ABB RobotStudio station: simulation.rsstn

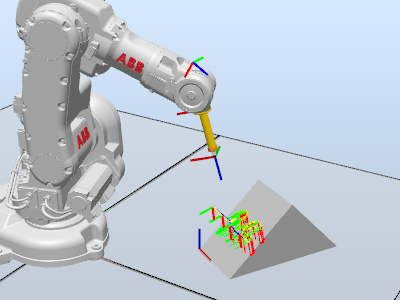
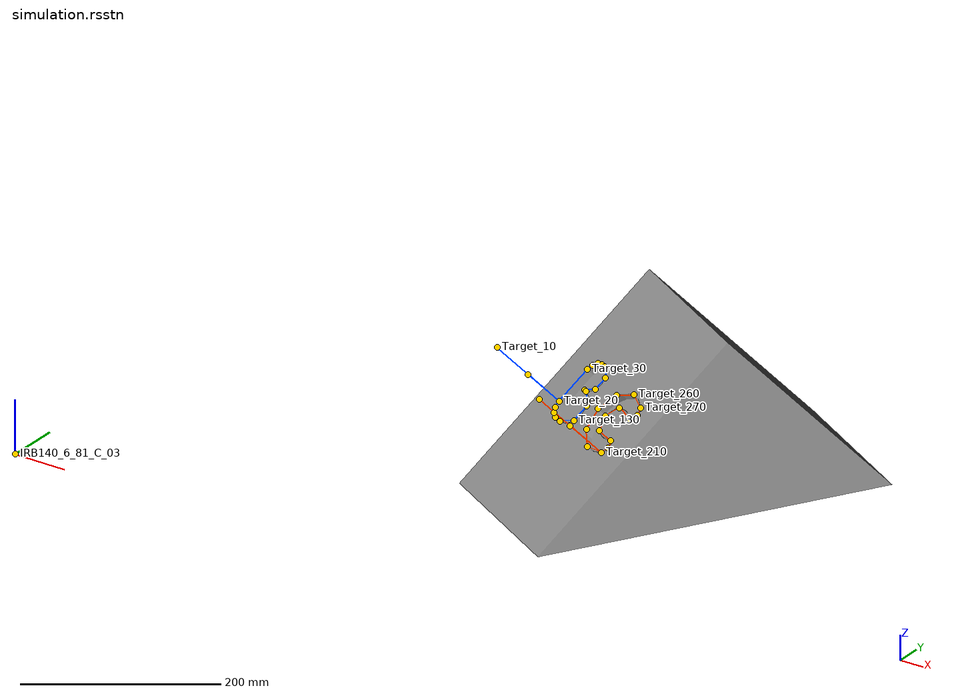
[picture v1: parts stored in the station drawn from their meshes, with robot base, taught points and paths (robot models come from the ABB library and are not in the file)]
Station simulation (saved by RobotStudio 22.2.9947.0)
Controller Controller7
  mechanical unit ROB_1: IRB140_6_81_C_03, 6 joints, base frame (0, 0, 0) mm
Layout (positions relative to the parent item):
  - IRB140_6_81_C_03 [mechanism, from Robots\IRB140_6_81_C_G_03.rslib] at (0, 0, 0) mm; joint values [0.3491, 0.0873, 0.3491, 0, 0.8727, 0] (rad or m)
  - MarkerTool [mechanism] at (434.7, 158.22, 487.25) mm, rotated rx 180 ry 15 rz -160 deg
      TCP MarkerTool at (0, 0, 145) mm
      links: ToolAssambly
  - Triangle [part] at (400, 200, 0) mm, rotated rx 0 ry 0 rz -30 deg, size 185 x 389.2 x 194.1 mm
Attachment: MarkerTool is attached to IRB140_6_81_C_03 / Link6
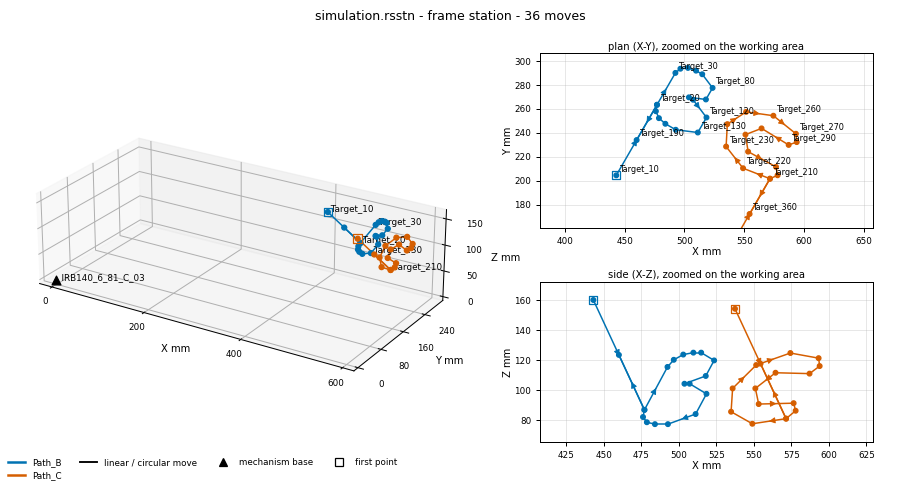
[picture p0: tool path of simulation.rsstn in frame station, 36 of 38 moves have a stored position in this frame; points joined in program order, loops and branches not executed]
Targets, tools, work objects and paths stored in the station, written as RAPID:
! task T_ROB1
MODULE CalibData
  PERS tooldata MarkerTool:=[TRUE,[[0,0,145],[1,0,0,0]],[0.1,[0,0,61],[1,0,0,0],0,0,0]];
  TASK PERS wobjdata Canvas:=[FALSE,TRUE,"",[[400.001,200,0],[0.9659258,0,0,-0.258819143]],[[0,0,0],[1,0,0,0]]];
ENDMODULE

! task T_ROB1
MODULE Module1
  CONST robtarget Target_10:=[[34.950823156,25.414242905,160.180640129],[0.35336537,-0.898969249,0.240877877,0.094683961],[0,0,0,0],[9E+09,9E+09,9E+09,9E+09,9E+09,9E+09]];
  CONST robtarget Target_20:=[[34.950809352,93.508617436,86.947067519],[0.35336537,-0.898969249,0.240877877,0.094683961],[0,0,0,0],[9E+09,9E+09,9E+09,9E+09,9E+09,9E+09]];
  CONST robtarget Target_30:=[[34.950803116,124.266717933,115.546704822],[0.35336537,-0.898969249,0.240877877,0.094683961],[0,0,0,0],[9E+09,9E+09,9E+09,9E+09,9E+09,9E+09]];
  CONST robtarget Target_40:=[[36.826446423,129.393068396,120.31331104],[0.353365369,-0.89896925,0.240877877,0.094683961],[0,0,0,0],[9E+09,9E+09,9E+09,9E+09,9E+09,9E+09]];
  CONST robtarget Target_50:=[[41.950801316,133.145818152,123.80270897],[0.35336537,-0.898969249,0.240877877,0.09468396],[0,0,0,0],[9E+09,9E+09,9E+09,9E+09,9E+09,9E+09]];
  CONST robtarget Target_60:=[[48.950801037,134.519420935,125.079917257],[0.35336537,-0.898969249,0.240877877,0.094683961],[0,0,0,0],[9E+09,9E+09,9E+09,9E+09,9E+09,9E+09]];
  CONST robtarget Target_70:=[[54.950801037,134.519422152,125.079917257],[0.35336537,-0.898969249,0.240877877,0.094683961],[0,0,0,0],[9E+09,9E+09,9E+09,9E+09,9E+09,9E+09]];
  CONST robtarget Target_80:=[[68.129449616,128.947305169,119.898823543],[0.35336537,-0.898969249,0.240877877,0.094683961],[0,0,0,0],[9E+09,9E+09,9E+09,9E+09,9E+09,9E+09]];
  CONST robtarget Target_90:=[[68.129451875,117.803065859,109.536636114],[0.353365369,-0.89896925,0.240877877,0.094683961],[0,0,0,0],[9E+09,9E+09,9E+09,9E+09,9E+09,9E+09]];
  CONST robtarget Target_100:=[[54.950805555,112.230943533,104.355542399],[0.35336537,-0.898969249,0.240877877,0.094683961],[0,0,0,0],[9E+09,9E+09,9E+09,9E+09,9E+09,9E+09]];
  CONST robtarget Target_110:=[[58.950805555,112.230944343,104.355542399],[0.35336537,-0.898969249,0.240877877,0.094683961],[0,0,0,0],[9E+09,9E+09,9E+09,9E+09,9E+09,9E+09]];
  CONST robtarget Target_120:=[[76.083048708,104.987192264,97.620120571],[0.35336537,-0.898969249,0.240877877,0.094683961],[0,0,0,0],[9E+09,9E+09,9E+09,9E+09,9E+09,9E+09]];
  CONST robtarget Target_130:=[[76.083051645,90.499681161,84.149276913],[0.353365369,-0.89896925,0.240877877,0.094683961],[0,0,0,0],[9E+09,9E+09,9E+09,9E+09,9E+09,9E+09]];
  CONST robtarget Target_140:=[[58.95081143,83.255922137,77.413855085],[0.35336537,-0.898969249,0.240877877,0.094683961],[0,0,0,0],[9E+09,9E+09,9E+09,9E+09,9E+09,9E+09]];
  CONST robtarget Target_150:=[[48.95081143,83.25592011,77.413855085],[0.35336537,-0.898969249,0.240877877,0.094683961],[0,0,0,0],[9E+09,9E+09,9E+09,9E+09,9E+09,9E+09]];
  CONST robtarget Target_160:=[[41.950811151,84.629520055,78.691063371],[0.35336537,-0.898969249,0.240877877,0.094683961],[0,0,0,0],[9E+09,9E+09,9E+09,9E+09,9E+09,9E+09]];
  CONST robtarget Target_170:=[[36.826454737,88.382267733,82.180461302],[0.35336537,-0.898969249,0.240877877,0.094683961],[0,0,0,0],[9E+09,9E+09,9E+09,9E+09,9E+09,9E+09]];
  CONST robtarget Target_180:=[[34.950809352,93.508617436,86.947067519],[0.35336537,-0.898969249,0.240877877,0.094683961],[0,0,0,0],[9E+09,9E+09,9E+09,9E+09,9E+09,9E+09]];
  CONST robtarget Target_190:=[[34.950816254,59.461430171,123.563853824],[0.35336537,-0.898969249,0.240877877,0.094683961],[0,0,0,0],[9E+09,9E+09,9E+09,9E+09,9E+09,9E+09]];
  CONST robtarget Target_200:=[[147.617491101,19.11128582,154.319974583],[0.35336537,-0.898969249,0.240877877,0.094683961],[0,0,0,0],[9E+09,9E+09,9E+09,9E+09,9E+09,9E+09]];
  CONST robtarget Target_210:=[[147.617477296,87.205660351,81.086401974],[0.35336537,-0.898969249,0.240877877,0.094683961],[0,0,0,0],[9E+09,9E+09,9E+09,9E+09,9E+09,9E+09]];
  CONST robtarget Target_220:=[[123.769810397,83.538318205,77.676421666],[0.35336537,-0.898969249,0.240877877,0.094683961],[0,0,0,0],[9E+09,9E+09,9E+09,9E+09,9E+09,9E+09]];
  CONST robtarget Target_230:=[[102.433503633,92.15845815,85.691643532],[0.35336537,-0.898969249,0.240877877,0.094683961],[0,0,0,0],[9E+09,9E+09,9E+09,9E+09,9E+09,9E+09]];
  CONST robtarget Target_240:=[[93.950806233,108.887679646,101.246886171],[0.35336537,-0.898969249,0.240877877,0.094683961],[0,0,0,0],[9E+09,9E+09,9E+09,9E+09,9E+09,9E+09]];
  CONST robtarget Target_250:=[[102.433496851,125.616904581,116.80212881],[0.35336537,-0.898969249,0.240877877,0.094683961],[0,0,0,0],[9E+09,9E+09,9E+09,9E+09,9E+09,9E+09]];
  CONST robtarget Target_260:=[[123.769800119,134.237053177,124.817350675],[0.353365369,-0.89896925,0.240877877,0.094683961],[0,0,0,0],[9E+09,9E+09,9E+09,9E+09,9E+09,9E+09]];
  CONST robtarget Target_270:=[[147.617468505,130.5697207,121.407370368],[0.35336537,-0.898969249,0.240877877,0.094683961],[0,0,0,0],[9E+09,9E+09,9E+09,9E+09,9E+09,9E+09]];
  CONST robtarget Target_280:=[[151.694170772,124.899768155,116.135308461],[0.35336537,-0.898969249,0.240877877,0.094683961],[0,0,0,0],[9E+09,9E+09,9E+09,9E+09,9E+09,9E+09]];
  CONST robtarget Target_290:=[[147.027505204,119.479259665,111.095187412],[0.35336537,-0.898969249,0.240877877,0.094683962],[0,0,0,0],[9E+09,9E+09,9E+09,9E+09,9E+09,9E+09]];
  CONST robtarget Target_300:=[[120.497500856,120.109201737,111.680928024],[0.35336537,-0.898969249,0.240877877,0.094683961],[0,0,0,0],[9E+09,9E+09,9E+09,9E+09,9E+09,9E+09]];
  CONST robtarget Target_310:=[[111.450806233,108.887683193,101.246886171],[0.35336537,-0.898969249,0.240877877,0.094683961],[0,0,0,0],[9E+09,9E+09,9E+09,9E+09,9E+09,9E+09]];
  CONST robtarget Target_320:=[[120.497505406,97.666168317,90.812844318],[0.35336537,-0.898969249,0.240877877,0.094683961],[0,0,0,0],[9E+09,9E+09,9E+09,9E+09,9E+09,9E+09]];
  CONST robtarget Target_330:=[[147.027509499,98.296121147,91.39858493],[0.353365371,-0.898969249,0.240877877,0.094683961],[0,0,0,0],[9E+09,9E+09,9E+09,9E+09,9E+09,9E+09]];
  CONST robtarget Target_340:=[[151.694177264,92.875614549,86.358463881],[0.35336537,-0.898969249,0.240877877,0.094683961],[0,0,0,0],[9E+09,9E+09,9E+09,9E+09,9E+09,9E+09]];
  CONST robtarget Target_350:=[[147.617477296,87.205660351,81.086401974],[0.35336537,-0.898969249,0.240877877,0.094683961],[0,0,0,0],[9E+09,9E+09,9E+09,9E+09,9E+09,9E+09]];
  CONST robtarget Target_360:=[[147.617484199,53.158473085,117.703188278],[0.35336537,-0.898969249,0.240877877,0.094683961],[0,0,0,0],[9E+09,9E+09,9E+09,9E+09,9E+09,9E+09]];
  CONST jointtarget Home:=[[0,0,0,0,30,0],[9E+09,9E+09,9E+09,9E+09,9E+09,9E+09]];
  CONST jointtarget Middle:=[[20,5,20,0,50,0],[9E+09,9E+09,9E+09,9E+09,9E+09,9E+09]];
  PROC Path_B()
    MoveL Target_10,v200,z50,MarkerTool\WObj:=Canvas;
    MoveL Target_20,v200,z50,MarkerTool\WObj:=Canvas;
    MoveL Target_30,v200,z50,MarkerTool\WObj:=Canvas;
    MoveL Target_40,v200,z50,MarkerTool\WObj:=Canvas;
    MoveL Target_50,v200,z50,MarkerTool\WObj:=Canvas;
    MoveL Target_60,v200,z50,MarkerTool\WObj:=Canvas;
    MoveL Target_70,v200,z50,MarkerTool\WObj:=Canvas;
    MoveL Target_80,v200,z50,MarkerTool\WObj:=Canvas;
    MoveL Target_90,v200,z50,MarkerTool\WObj:=Canvas;
    MoveL Target_100,v200,z50,MarkerTool\WObj:=Canvas;
    MoveL Target_110,v200,z50,MarkerTool\WObj:=Canvas;
    MoveL Target_120,v200,z50,MarkerTool\WObj:=Canvas;
    MoveL Target_130,v200,z50,MarkerTool\WObj:=Canvas;
    MoveL Target_140,v200,z50,MarkerTool\WObj:=Canvas;
    MoveL Target_150,v200,z50,MarkerTool\WObj:=Canvas;
    MoveL Target_160,v200,z50,MarkerTool\WObj:=Canvas;
    MoveL Target_170,v200,z50,MarkerTool\WObj:=Canvas;
    MoveL Target_180,v200,z50,MarkerTool\WObj:=Canvas;
    MoveL Target_190,v200,z50,MarkerTool\WObj:=Canvas;
  ENDPROC
  PROC Path_C()
    MoveL Target_200,v200,z50,MarkerTool\WObj:=Canvas;
    MoveL Target_210,v200,z50,MarkerTool\WObj:=Canvas;
    MoveL Target_220,v200,z50,MarkerTool\WObj:=Canvas;
    MoveL Target_230,v200,z50,MarkerTool\WObj:=Canvas;
    MoveL Target_240,v200,z50,MarkerTool\WObj:=Canvas;
    MoveL Target_250,v200,z50,MarkerTool\WObj:=Canvas;
    MoveL Target_260,v200,z50,MarkerTool\WObj:=Canvas;
    MoveL Target_270,v200,z50,MarkerTool\WObj:=Canvas;
    MoveL Target_280,v200,z50,MarkerTool\WObj:=Canvas;
    MoveL Target_290,v200,z50,MarkerTool\WObj:=Canvas;
    MoveL Target_300,v200,z50,MarkerTool\WObj:=Canvas;
    MoveL Target_310,v200,z50,MarkerTool\WObj:=Canvas;
    MoveL Target_320,v200,z50,MarkerTool\WObj:=Canvas;
    MoveL Target_330,v200,z50,MarkerTool\WObj:=Canvas;
    MoveL Target_340,v200,z50,MarkerTool\WObj:=Canvas;
    MoveL Target_350,v200,z50,MarkerTool\WObj:=Canvas;
    MoveL Target_360,v200,z50,MarkerTool\WObj:=Canvas;
  ENDPROC
  PROC Path_Home()
    MoveAbsJ Home,v1000,z100,MarkerTool\WObj:=Canvas;
  ENDPROC
  PROC Path_Middle()
    MoveAbsJ Middle,v1000,z100,MarkerTool\WObj:=Canvas;
  ENDPROC
ENDMODULE

